TYPE Int_2Byte :
UNION
	sValue			:INT; 
	arrByte 		:ARRAY[0..1] OF BYTE;
END_UNION
END_TYPE

(* stored: Version 1.1.0.1
   DUT Int_2Byte: Id {4fbd5857-01aa-4d0e-acf1-baf99d09c829} *)
